// Parses a 32-bit little-endian integer.
FUNCTION F_ParseRawLittleEndian32 : HRESULT
VAR_IN_OUT      
    stCtx : ST_ParseContext;
END_VAR
VAR_OUTPUT
    nValue : UDINT;
END_VAR
VAR CONSTANT
    cLength : UDINT := SIZEOF(nValue);
END_VAR


F_ParseRawLittleEndian32 := F_ReadFromBuffer(stCtx, F_ToAnyType(nValue), cLength);

END_FUNCTION

(* stored: Version 1.1.0.1
   POU F_ParseRawLittleEndian32: Id {562fac10-4f40-4f06-ac41-d13ff8cdd378}, SpecialFunc None *)
